(* IEC 61131-3 sources: SRCI/RobotLibrary/RobotLibrary/Functions/Common, 2 files *)

(* ---- CheckTimeout.st ---- *)
FUNCTION CheckTimeout : DINT
VAR_INPUT
  /// Reference to TON instance
  rTimer : REFERENCE TO TON;
END_VAR

  // Call timer
  rTimer();

  // check if timer elapsed
  IF (rTimer.Q = TRUE)
  THEN
    // assign return value
    CheckTimeout := RobotLibraryConstants.OK;
  ELSE
    // assign return value
    CheckTimeout := RobotLibraryConstants.RUNNING;
  END_IF

END_FUNCTION

(* ---- SetTimeout.st ---- *)
FUNCTION SetTimeout : DINT
VAR_INPUT
  /// Timeout to be set
  PT     : TIME;
  /// Reference to TON instance
  rTimer : REFERENCE TO TON;
END_VAR

  rTimer(IN := FALSE);          // Reset timer
  rTimer(PT := PT, IN := TRUE); // Start timer

  // assign return value
  SetTimeout := RobotLibraryConstants.OK;

END_FUNCTION
